{attribute 'qualified_only'}
VAR_GLOBAL
	// UI Command
	bRun: BOOL := FALSE;
	// UI Indicator
	bIsRunning: BOOL := FALSE;
	nProgress: USINT := 0;
	
	// bErrors: BOOL := FALSE;
END_VAR

(* stored: Version 1.1.0.1, ProductVersion 3.1.4024.3
   GVL GVL_Control: Id {804ca955-0c89-4f28-b6c5-be1d13de4a28} *)
